FUNCTION_BLOCK NextFeedHorizonCalc (* Basic Function Block Type *)
  (* Standard: 61499-2 *)
  (* Version 0.0, 7/15/2026, Schneider Electric, Template *)
  PACKAGE SE.Nereda;
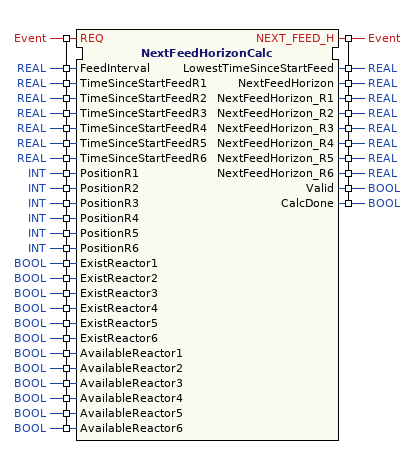
  EVENT_INPUT
    REQ WITH FeedInterval, TimeSinceStartFeedR1, TimeSinceStartFeedR2, TimeSinceStartFeedR3, TimeSinceStartFeedR4, TimeSinceStartFeedR5, TimeSinceStartFeedR6, PositionR1, PositionR2, PositionR3, PositionR4, PositionR5, PositionR6, ExistReactor1, ExistReactor2, ExistReactor3, ExistReactor4, ExistReactor5, ExistReactor6, AvailableReactor1, AvailableReactor2, AvailableReactor3, AvailableReactor4, AvailableReactor5, AvailableReactor6;
  END_EVENT
  EVENT_OUTPUT
    NEXT_FEED_H WITH NextFeedHorizon, Valid, NextFeedHorizon_R2, NextFeedHorizon_R3, NextFeedHorizon_R4, NextFeedHorizon_R5, NextFeedHorizon_R1, LowestTimeSinceStartFeed, NextFeedHorizon_R6, CalcDone;
  END_EVENT
  VAR_INPUT
    FeedInterval : REAL;
    TimeSinceStartFeedR1 : REAL;
    TimeSinceStartFeedR2 : REAL;
    TimeSinceStartFeedR3 : REAL;
    TimeSinceStartFeedR4 : REAL;
    TimeSinceStartFeedR5 : REAL;
    TimeSinceStartFeedR6 : REAL;
    PositionR1 : INT;
    PositionR2 : INT;
    PositionR3 : INT;
    PositionR4 : INT;
    PositionR5 : INT;
    PositionR6 : INT;
    ExistReactor1 : BOOL;
    ExistReactor2 : BOOL;
    ExistReactor3 : BOOL;
    ExistReactor4 : BOOL;
    ExistReactor5 : BOOL;
    ExistReactor6 : BOOL;
    AvailableReactor1 : BOOL;
    AvailableReactor2 : BOOL;
    AvailableReactor3 : BOOL;
    AvailableReactor4 : BOOL;
    AvailableReactor5 : BOOL;
    AvailableReactor6 : BOOL;
  END_VAR
  VAR_OUTPUT
    LowestTimeSinceStartFeed : REAL;
    NextFeedHorizon : REAL;
    NextFeedHorizon_R1 : REAL;
    NextFeedHorizon_R2 : REAL;
    NextFeedHorizon_R3 : REAL;
    NextFeedHorizon_R4 : REAL;
    NextFeedHorizon_R5 : REAL;
    NextFeedHorizon_R6 : REAL;
    Valid : BOOL;
    CalcDone : BOOL;
  END_VAR
  VAR
    TimeSinceStartFeed : REAL;
    FirstValueFound : BOOL;
    R1Used : BOOL;
    R2Used : BOOL;
    R3Used : BOOL;
    R4Used : BOOL;
    R5Used : BOOL;
    R6Used : BOOL;
  END_VAR
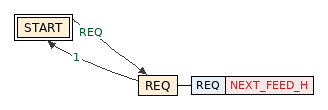
  EC_STATES
    START; (* Initial State *)
    REQ : REQ -> NEXT_FEED_H; (* Normal execution *)
  END_STATES
  EC_TRANSITIONS
    START TO REQ := REQ;
    REQ TO START := 1;
  END_TRANSITIONS
  ALGORITHM REQ IN ST: (* Normally executed algorithm *)
;
R1Used := ExistReactor1 AND AvailableReactor1;
R2Used := ExistReactor2 AND AvailableReactor2;
R3Used := ExistReactor3 AND AvailableReactor3;
R4Used := ExistReactor4 AND AvailableReactor4;
R5Used := ExistReactor5 AND AvailableReactor5;
R6Used := ExistReactor6 AND AvailableReactor6;

Valid := FALSE;
FirstValueFound := FALSE;
LowestTimeSinceStartFeed := 0;
NextFeedHorizon := 0;

NextFeedHorizon_R1 := 0;
NextFeedHorizon_R2 := 0;
NextFeedHorizon_R3 := 0;
NextFeedHorizon_R4 := 0;
NextFeedHorizon_R5 := 0;
NextFeedHorizon_R6 := 0;

IF R1Used THEN
	LowestTimeSinceStartFeed := TimeSinceStartFeedR1;
	FirstValueFound := TRUE;
END_IF;

IF R2Used THEN
	IF NOT FirstValueFound THEN
		LowestTimeSinceStartFeed := TimeSinceStartFeedR2;
		FirstValueFound := TRUE;
	ELSIF TimeSinceStartFeedR2 < LowestTimeSinceStartFeed THEN
		LowestTimeSinceStartFeed := TimeSinceStartFeedR2;
	END_IF;
END_IF;

IF R3Used THEN
	IF NOT FirstValueFound THEN
		LowestTimeSinceStartFeed := TimeSinceStartFeedR3;
		FirstValueFound := TRUE;
	ELSIF TimeSinceStartFeedR3 < LowestTimeSinceStartFeed THEN
		LowestTimeSinceStartFeed := TimeSinceStartFeedR3;
	END_IF;
END_IF;

IF R4Used THEN
	IF NOT FirstValueFound THEN
		LowestTimeSinceStartFeed := TimeSinceStartFeedR4;
		FirstValueFound := TRUE;
	ELSIF TimeSinceStartFeedR4 < LowestTimeSinceStartFeed THEN
		LowestTimeSinceStartFeed := TimeSinceStartFeedR4;
	END_IF;
END_IF;

IF R5Used THEN
	IF NOT FirstValueFound THEN
		LowestTimeSinceStartFeed := TimeSinceStartFeedR5;
		FirstValueFound := TRUE;
	ELSIF TimeSinceStartFeedR5 < LowestTimeSinceStartFeed THEN
		LowestTimeSinceStartFeed := TimeSinceStartFeedR5;
	END_IF;
END_IF;

IF R6Used THEN
	IF NOT FirstValueFound THEN
		LowestTimeSinceStartFeed := TimeSinceStartFeedR6;
		FirstValueFound := TRUE;
	ELSIF TimeSinceStartFeedR6 < LowestTimeSinceStartFeed THEN
		LowestTimeSinceStartFeed := TimeSinceStartFeedR6;
	END_IF;
END_IF;

Valid := FirstValueFound AND (FeedInterval > 0);

IF Valid THEN
	IF LowestTimeSinceStartFeed >= FeedInterval THEN
		NextFeedHorizon := 0;
	ELSE
		NextFeedHorizon := FeedInterval - LowestTimeSinceStartFeed;
	END_IF;

	IF R1Used THEN
		NextFeedHorizon_R1 := NextFeedHorizon + (PositionR1 - 1) * FeedInterval;
	END_IF;

	IF R2Used THEN
		NextFeedHorizon_R2 := NextFeedHorizon + (PositionR2 - 1) * FeedInterval;
	END_IF;

	IF R3Used THEN
		NextFeedHorizon_R3 := NextFeedHorizon + (PositionR3 - 1) * FeedInterval;
	END_IF;

	IF R4Used THEN
		NextFeedHorizon_R4 := NextFeedHorizon + (PositionR4 - 1) * FeedInterval;
	END_IF;

	IF R5Used THEN
		NextFeedHorizon_R5 := NextFeedHorizon + (PositionR5 - 1) * FeedInterval;
	END_IF;

	IF R6Used THEN
		NextFeedHorizon_R6 := NextFeedHorizon + (PositionR6 - 1) * FeedInterval;
	END_IF;
END_IF;

CalcDone := Valid AND  AND
		(AvailableReactor1 AND NextFeedHorizon_R1 <> 0 OR
		AvailableReactor2 AND NextFeedHorizon_R2 <> 0 OR
		AvailableReactor3 AND NextFeedHorizon_R3 <> 0 OR
		AvailableReactor4 AND NextFeedHorizon_R4 <> 0 OR
		AvailableReactor5 AND NextFeedHorizon_R5 <> 0 OR
		AvailableReactor6 AND NextFeedHorizon_R6 <> 0);
  END_ALGORITHM
END_FUNCTION_BLOCK
